TYPE ST_SignalTower :
STRUCT
	Lamp_Green : BOOL;
	Lamp_Yellow : BOOL;
	Lamp_Red	: BOOL;
	Buzz		: BOOL;
END_STRUCT
END_TYPE

(* stored: Version 1.1.0.1, ProductVersion 3.1.4024.13
   DUT ST_SignalTower: Id {40a89c78-bc7c-43a2-b692-3296f387a2e8} *)
